{attribute 'pack_mode' := '1'}
    {attribute 'OPC.UA.DA' := '1'}
    {attribute 'OPC.UA.DA.StructuredType' := '1'}
    (*
    ST_RW_Motor_Starter_Hybrid_New_HMI_IgnitionExp
    ==================================================
    Generated from Ignition UDT: RW_Motor_Starter_Hybrid_New
    Total tags: 51
    Generated on: 2025-09-16 11:33:46
    *)
    TYPE ST_RW_Motor_Starter_Hybrid_New_HMI_IgnitionExp :
    STRUCT
        {attribute 'OPC.UA.DA' := '1'}
        Run_Feedback : BOOL := FALSE;
        {attribute 'OPC.UA.DA' := '1'}
        Manual_Cmd : BOOL := FALSE;
        {attribute 'OPC.UA.DA' := '1'}
        Disconnect_Alarm : BOOL := FALSE;
        {attribute 'OPC.UA.DA' := '1'}
        Starter_Faulted : BOOL := FALSE;
        {attribute 'OPC.UA.DA' := '1'}
        Disconnect_Enable : BOOL := FALSE;

        {attribute 'OPC.UA.DA' := '1'}
        Feedback_Mismatch_Alarm : BOOL := FALSE;
        {attribute 'OPC.UA.DA' := '1'}
        Starter_Ready : BOOL := FALSE;
        {attribute 'OPC.UA.DA' := '1'}
        Voltage_OK : BOOL := FALSE;
        {attribute 'OPC.UA.DA' := '1'}
        Running : BOOL := FALSE;
        {attribute 'OPC.UA.DA' := '1'}
        Asset_Alarm : BOOL := FALSE;

        {attribute 'OPC.UA.DA' := '1'}
        Disconnect : BOOL := FALSE;
        {attribute 'OPC.UA.DA' := '1'}
        {attribute 'OPC.UA.DA.Access' := '1'}
        Interlock_Tripped : BOOL := FALSE;		// Read-only tag
        {attribute 'OPC.UA.DA' := '1'}
        Feedback_Mismatch_Alarm_Timer : LREAL := 0.0;
        {attribute 'OPC.UA.DA' := '1'}
        Motor_Current : REAL := 0.0;
        Interlocks_Interlock_24 : ST_RW_Interlock_Equipment_Map_HMI_IgnitionExp;		// UDT Instance: Interlock 24 (Redwood/RW_Interlock_Equipment_Map)

        Interlocks_Interlock_4 : ST_RW_Interlock_Equipment_Map_HMI_IgnitionExp;		// UDT Instance: Interlock 4 (Redwood/RW_Interlock_Equipment_Map)
        Interlocks_Interlock_27 : ST_RW_Interlock_Equipment_Map_HMI_IgnitionExp;		// UDT Instance: Interlock 27 (Redwood/RW_Interlock_Equipment_Map)
        Interlocks_Interlock_30 : ST_RW_Interlock_Equipment_Map_HMI_IgnitionExp;		// UDT Instance: Interlock 30 (Redwood/RW_Interlock_Equipment_Map)
        Interlocks_Interlock_14 : ST_RW_Interlock_Equipment_Map_HMI_IgnitionExp;		// UDT Instance: Interlock 14 (Redwood/RW_Interlock_Equipment_Map)
        Interlocks_Interlock_5 : ST_RW_Interlock_Equipment_Map_HMI_IgnitionExp;		// UDT Instance: Interlock 5 (Redwood/RW_Interlock_Equipment_Map)

        Interlocks_Interlock_21 : ST_RW_Interlock_Equipment_Map_HMI_IgnitionExp;		// UDT Instance: Interlock 21 (Redwood/RW_Interlock_Equipment_Map)
        Interlocks_Interlock_1 : ST_RW_Interlock_Equipment_Map_HMI_IgnitionExp;		// UDT Instance: Interlock 1 (Redwood/RW_Interlock_Equipment_Map)
        Interlocks_Interlock_10 : ST_RW_Interlock_Equipment_Map_HMI_IgnitionExp;		// UDT Instance: Interlock 10 (Redwood/RW_Interlock_Equipment_Map)
        Interlocks_Interlock_7 : ST_RW_Interlock_Equipment_Map_HMI_IgnitionExp;		// UDT Instance: Interlock 7 (Redwood/RW_Interlock_Equipment_Map)
        Interlocks_Interlock_9 : ST_RW_Interlock_Equipment_Map_HMI_IgnitionExp;		// UDT Instance: Interlock 9 (Redwood/RW_Interlock_Equipment_Map)

        Interlocks_Interlock_17 : ST_RW_Interlock_Equipment_Map_HMI_IgnitionExp;		// UDT Instance: Interlock 17 (Redwood/RW_Interlock_Equipment_Map)
        Interlocks_Interlock_15 : ST_RW_Interlock_Equipment_Map_HMI_IgnitionExp;		// UDT Instance: Interlock 15 (Redwood/RW_Interlock_Equipment_Map)
        Interlocks_Interlock_28 : ST_RW_Interlock_Equipment_Map_HMI_IgnitionExp;		// UDT Instance: Interlock 28 (Redwood/RW_Interlock_Equipment_Map)
        Interlocks_Interlock_3 : ST_RW_Interlock_Equipment_Map_HMI_IgnitionExp;		// UDT Instance: Interlock 3 (Redwood/RW_Interlock_Equipment_Map)
        Interlocks_Interlock_22 : ST_RW_Interlock_Equipment_Map_HMI_IgnitionExp;		// UDT Instance: Interlock 22 (Redwood/RW_Interlock_Equipment_Map)

        Interlocks_Interlock_12 : ST_RW_Interlock_Equipment_Map_HMI_IgnitionExp;		// UDT Instance: Interlock 12 (Redwood/RW_Interlock_Equipment_Map)
        Interlocks_Interlock_29 : ST_RW_Interlock_Equipment_Map_HMI_IgnitionExp;		// UDT Instance: Interlock 29 (Redwood/RW_Interlock_Equipment_Map)
        Interlocks_Interlock_31 : ST_RW_Interlock_Equipment_Map_HMI_IgnitionExp;		// UDT Instance: Interlock 31 (Redwood/RW_Interlock_Equipment_Map)
        Interlocks_Interlock_23 : ST_RW_Interlock_Equipment_Map_HMI_IgnitionExp;		// UDT Instance: Interlock 23 (Redwood/RW_Interlock_Equipment_Map)
        Interlocks_Interlock_16 : ST_RW_Interlock_Equipment_Map_HMI_IgnitionExp;		// UDT Instance: Interlock 16 (Redwood/RW_Interlock_Equipment_Map)

        Interlocks_Interlock_6 : ST_RW_Interlock_Equipment_Map_HMI_IgnitionExp;		// UDT Instance: Interlock 6 (Redwood/RW_Interlock_Equipment_Map)
        Interlocks_Interlock_26 : ST_RW_Interlock_Equipment_Map_HMI_IgnitionExp;		// UDT Instance: Interlock 26 (Redwood/RW_Interlock_Equipment_Map)
        Interlocks_Interlock_11 : ST_RW_Interlock_Equipment_Map_HMI_IgnitionExp;		// UDT Instance: Interlock 11 (Redwood/RW_Interlock_Equipment_Map)
        Interlocks_Interlock_2 : ST_RW_Interlock_Equipment_Map_HMI_IgnitionExp;		// UDT Instance: Interlock 2 (Redwood/RW_Interlock_Equipment_Map)
        Interlocks_Interlock_19 : ST_RW_Interlock_Equipment_Map_HMI_IgnitionExp;		// UDT Instance: Interlock 19 (Redwood/RW_Interlock_Equipment_Map)

        Interlocks_Interlock_20 : ST_RW_Interlock_Equipment_Map_HMI_IgnitionExp;		// UDT Instance: Interlock 20 (Redwood/RW_Interlock_Equipment_Map)
        Interlocks_Interlock_13 : ST_RW_Interlock_Equipment_Map_HMI_IgnitionExp;		// UDT Instance: Interlock 13 (Redwood/RW_Interlock_Equipment_Map)
        Interlocks_Interlock_18 : ST_RW_Interlock_Equipment_Map_HMI_IgnitionExp;		// UDT Instance: Interlock 18 (Redwood/RW_Interlock_Equipment_Map)
        Interlocks_Interlock_25 : ST_RW_Interlock_Equipment_Map_HMI_IgnitionExp;		// UDT Instance: Interlock 25 (Redwood/RW_Interlock_Equipment_Map)
        Interlocks_Interlock_8 : ST_RW_Interlock_Equipment_Map_HMI_IgnitionExp;		// UDT Instance: Interlock 8 (Redwood/RW_Interlock_Equipment_Map)

        {attribute 'OPC.UA.DA' := '1'}
        Communication_Error : BOOL := FALSE;
        {attribute 'OPC.UA.DA' := '1'}
        Runtime_Counter : SINT := 0;
        {attribute 'OPC.UA.DA' := '1'}
        Manual_Mode : BOOL := FALSE;
        {attribute 'OPC.UA.DA' := '1'}
        Fault_Reset : BOOL := FALSE;
        {attribute 'OPC.UA.DA' := '1'}
        Command : BOOL := FALSE;

        {attribute 'OPC.UA.DA' := '1'}
        Runtime_Counter_Reset : BOOL := FALSE;
    END_STRUCT
    END_TYPE

(* stored: Version 1.1.0.1
   DUT ST_RW_Motor_Starter_Hybrid_New_HMI_IgnitionExp: Id {ef944859-2e1a-464b-8074-664b8b9a409d} *)
